(* Schneider Machine Expert - Basic project Star Delta Motor 3Phase, file version 1.7.0.0 *)
(* ProjectInformations: Name=New project *)

HARDWARE
  Cpu 0: TM221ME16R/G
  EthernetConfiguration: NetworkName=M221, IpAllocationMode=FixedAddress, IpAddress=0.0.0.0, SubnetMask=0.0.0.0
  SerialLineConfiguration: Baud=Baud19200, Parity=ParityEven, DataBits=DataBits8, StopBits=StopBits1, PhysicalMedium=PhysicalMediumRs485, TransmissionMode=TransmissionModeModbusRtu, SlaveId=1, Addressing=SlaveAddressing
  MastTask: UsePeriodScanMode=false, PeriodScan=100
  FastTask: Period=255
  CpuBehavior: StartingMode=StartAsPreviousState, AutoSaveRamOnEeprom=true, WatchdogPeriod=250

SYMBOLS  (address, symbol, comment, settings)
  %TM0        [Preset=5, Base=OneSecond]
  %I0.0     PB1
  %I0.1     PB2
  %I0.2     EMERGENCY
  %I0.3     TOR
  %Q0.0     K1M
  %Q0.1     L1
  %Q0.2     L2

POU New POU
  (* SectionNumber=1 *)

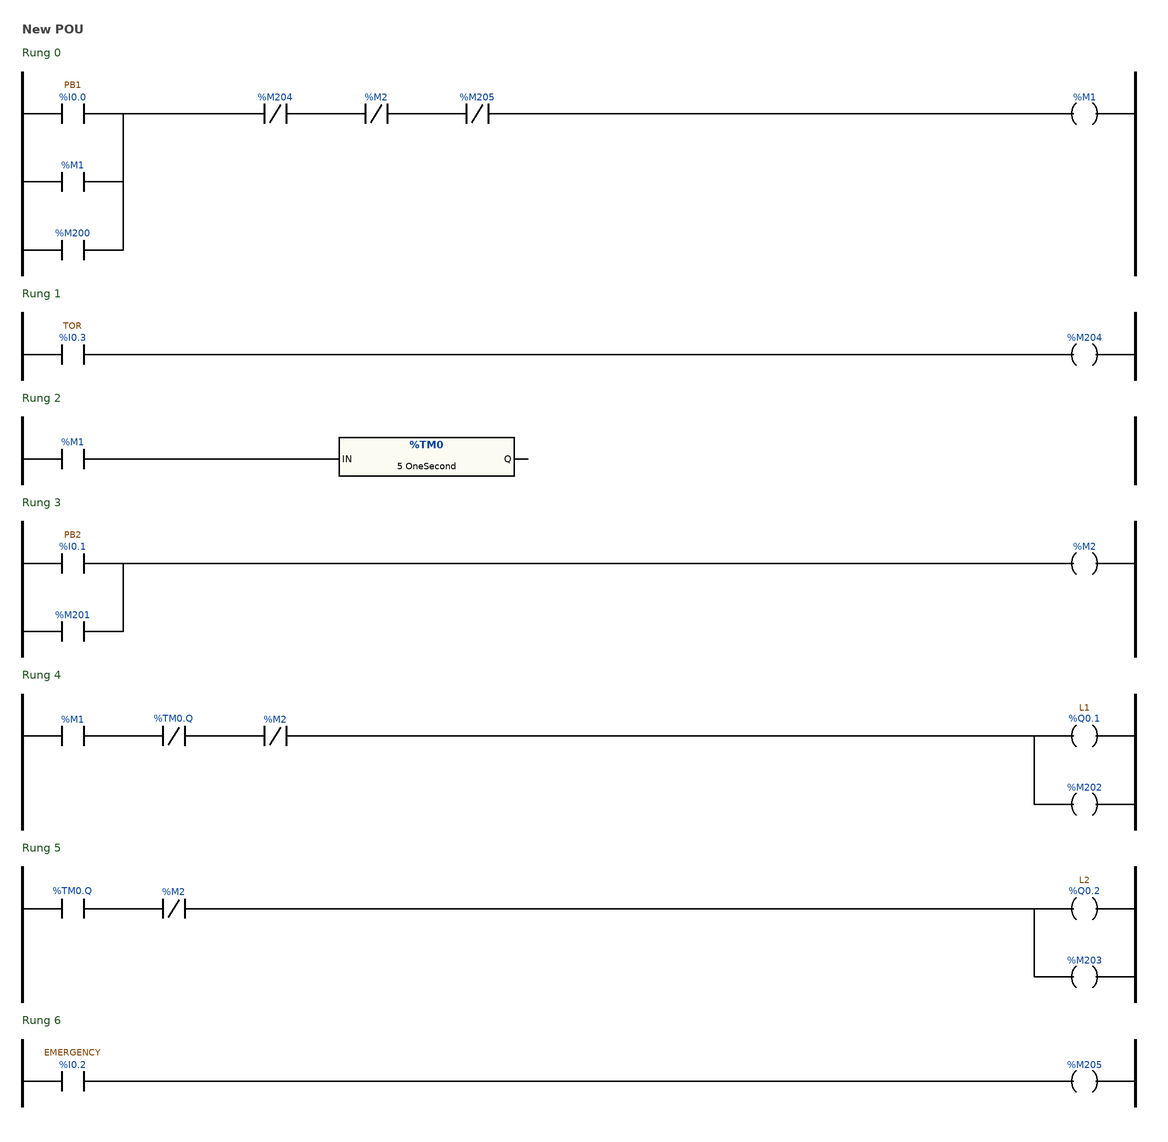

// Rung 0
  LD %I0.0                (* PB1 *)
  OR %M1
  OR %M200
  ANDN %M204
  ANDN %M2
  ANDN %M205
  ST %M1
  // as ST:
  //   %M1 := (PB1 OR %M1 OR %M200) AND NOT %M204 AND NOT %M2 AND NOT %M205;

// Rung 1
  LD %I0.3                (* TOR *)
  ST %M204
  // as ST:
  //   %M204 := TOR;

// Rung 2
  BLK %TM0
  LD %M1
  IN
  END_BLK
  // as ST:
  //   %TM0(IN := %M1);

// Rung 3
  LD %I0.1                (* PB2 *)
  OR %M201
  ST %M2
  // as ST:
  //   %M2 := PB2 OR %M201;

// Rung 4
  LD %M1
  ANDN %TM0.Q
  ANDN %M2
  ST %Q0.1                (* L1 *)
  ST %M202
  // as ST:
  //   L1 := %M1 AND NOT %TM0.Q AND NOT %M2;
  //   %M202 := %M1 AND NOT %TM0.Q AND NOT %M2;

// Rung 5
  LD %TM0.Q
  ANDN %M2
  ST %Q0.2                (* L2 *)
  ST %M203
  // as ST:
  //   L2 := %TM0.Q AND NOT %M2;
  //   %M203 := %TM0.Q AND NOT %M2;

// Rung 6
  LD %I0.2                (* EMERGENCY *)
  ST %M205
  // as ST:
  //   %M205 := EMERGENCY;
